Fanuc KAREL source: kb00022.KL

PROGRAM KB00022
%STACKSIZE=65535
%PRIORITY=65535
%NOLOCKGROUP
VAR
P1 : INTEGER
BEGIN
P1=1
CLEAR_SEMA(P1)
END KB00022
